(* Schneider Machine Expert - Basic project simple-water tank-level-from-uptomation-yt, file version 2.7.0.0 *)
(* ProjectInformations: Name=New project *)

HARDWARE
  Cpu 0: TM221M16R/G
  EthernetConfiguration: NetworkName=M221, IpAllocationMode=FixedAddress, IpAddress=0.0.0.0, SubnetMask=0.0.0.0
  SerialLineConfiguration: Baud=Baud19200, Parity=ParityEven, DataBits=DataBits8, StopBits=StopBits1, PhysicalMedium=PhysicalMediumRs485, TransmissionMode=TransmissionModeModbusRtu, SlaveId=1, Addressing=SlaveAddressing
  MastTask: UsePeriodScanMode=false, PeriodScan=100
  FastTask: Period=255
  CpuBehavior: StartingMode=StartAsPreviousState, AutoSaveRamOnEeprom=true, WatchdogPeriod=250

SYMBOLS  (address, symbol, comment, settings)
  %I0.0     STARTED
  %I0.1     LLS_TANK
  %I0.2     HLS_TANK
  %I0.3     LLS_POOL
  %I0.7     STOP
  %Q0.0     PUMP

POU New POU
  (* SectionNumber=1 *)

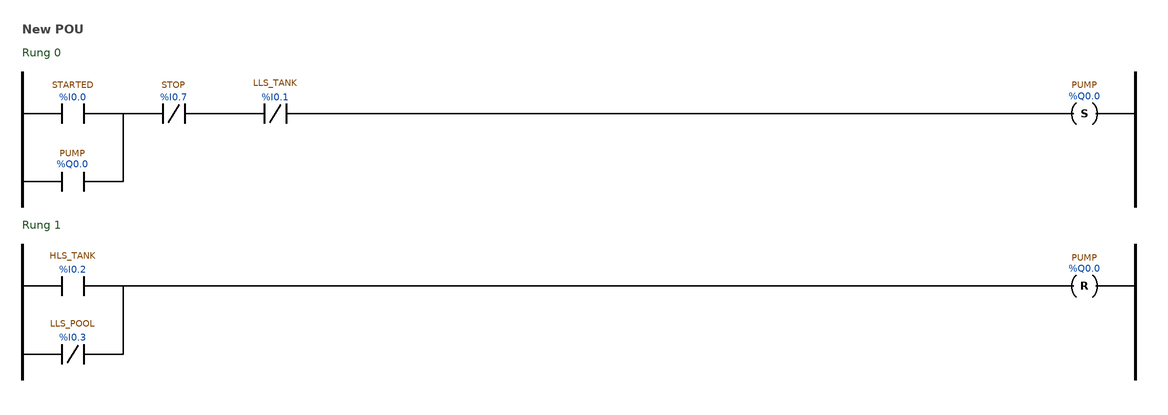

// Rung 0
  LD %I0.0                (* STARTED *)
  OR %Q0.0                (* PUMP *)
  ANDN %I0.7              (* STOP *)
  ANDN %I0.1              (* LLS_TANK *)
  S %Q0.0                 (* PUMP *)
  // as ST:
  //   IF (STARTED OR PUMP) AND NOT STOP AND NOT LLS_TANK THEN PUMP := TRUE; END_IF;

// Rung 1
  LD %I0.2                (* HLS_TANK *)
  ORN %I0.3               (* LLS_POOL *)
  R %Q0.0                 (* PUMP *)
  // as ST:
  //   IF HLS_TANK OR NOT LLS_POOL THEN PUMP := FALSE; END_IF;
